// TIA Portal V18 export
FUNCTION "IV3" : Void   // FC2100, LAD
{ S7_Optimized_Access := 'TRUE' }
VERSION : 0.1
// stored: AutoNumber false, IsIECCheckEnabled false, SetENOAutomatically false, UDAEnableTagReadback false
BEGIN

REGION Network 1: IV3
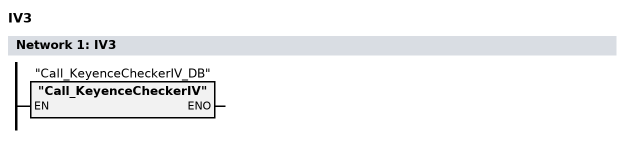
   RUNG wire#powerrail
      "Call_KeyenceCheckerIV_DB"()
   END_RUNG
   // the same network as SCL:
   "Call_KeyenceCheckerIV_DB"();   // "Call_KeyenceCheckerIV"
END_REGION
END_FUNCTION
